PROGRAM MAIN
VAR
	Counter AT %Q* : UDINT;
	In_1	AT %I* : UDINT;
	In_2	AT %I* : UDINT;
	
	{attribute 'TcInitSymbol'}
	TimeToConsume :UDINT:=10;
END_VAR

F_ConsumeTime(TimeToConsume);
Counter := (Counter + 1) MOD 200;

END_PROGRAM

(* stored: Version 1.1.0.1, ProductVersion 3.1.4026.18
   POU MAIN: Id {008ff7e3-702c-4b23-834b-f8aafcce3fa4}, SpecialFunc None *)
